Universal Robots PolyScope program: washer_wash_cup.urp

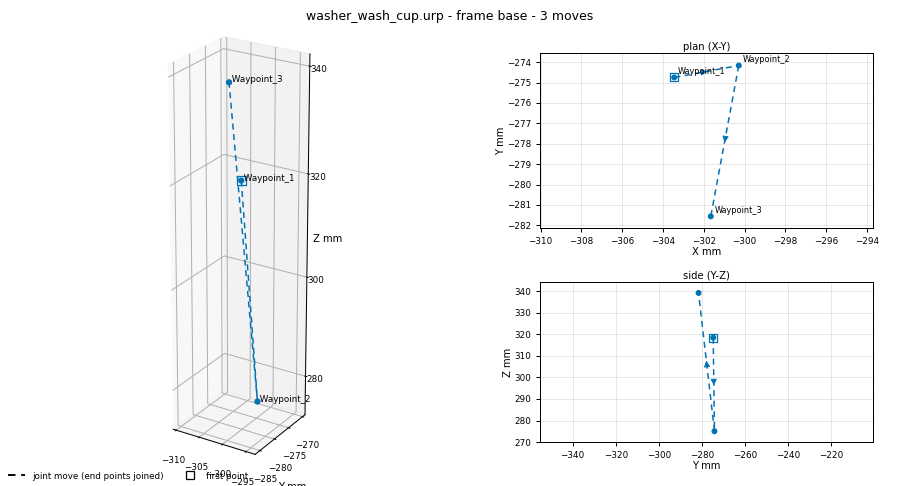
[picture p0: tool path of washer_wash_cup.urp in frame base, 3 of 3 moves have a stored position in this frame; points joined in program order, loops and branches not executed]
Program washer_wash_cup (installation=default directory=/programs createdIn=5.9.5.1031259 lastSavedIn=5.9.5.1031259 robotSerialNumber=20215500597)
Calibrated DH parameters: a=[0.000193, -0.066673, -0.391568, -0.000012, 0.00005, 0]; d=[0.162643, -472.05677, 465.132521, 7.058239, 0.099746, 0.099582]; alpha=[1.571116, 0.00089, 0.003862, 1.569269, -1.569248, 0]; deltaTheta=[0, -1.413394, 7.628392, 0.068187, 0, -0.000001]
Robot Program (runOnlyOnce=false)
  MoveJ speed 60 deg/s, acceleration 80 deg/s^2 (useActiveTCP=true) feature=Base
    Waypoint Waypoint_1: TCP in base x=-303.447 y=-274.748 z=318.451 mm, rx=1.141 ry=-1.1596 rz=1.2576 rad; joints [330.945, -97.077, 126.286, 340.772, -29.277, -277.9] deg; TCP offset x=0 y=0 z=191.5 mm, rx=0 ry=0 rz=0 rad
    Waypoint Waypoint_2: TCP in base x=-300.285 y=-274.165 z=275.036 mm, rx=1.2249 ry=-1.1919 rz=1.2251 rad; joints [331.056, -97.073, 129.567, 328.304, -30.165, -270.969] deg
    Wait Sleep waitTime=10
    Waypoint Waypoint_3: TCP in base x=-301.655 y=-281.558 z=339.221 mm, rx=1.1718 ry=-1.2852 rz=1.261 rad; joints [331.697, -104.003, 123.671, 339.068, -27.885, -264] deg
    Halt
